(* IEC 61131-3 sources: AXOpen/src/showcase/app/src/ComponentsDukaneWelders/Documentation, 1 file *)

(* ---- DocumentationContext.st ---- *)
NAMESPACE AXOpen.Components.Dukane.Welders
    {S7.extern=ReadWrite}
    CLASS DocumentationContext EXTENDS AXOpen.Core.AxoObject
        VAR PUBLIC
            rootObject      : AxoObject;
            componentOne    : AXOpen.Components.Dukane.Welders.Component_1;
            componentTwo    : AXOpen.Components.Dukane.Welders.Component_2;
        END_VAR

        METHOD PUBLIC Execute
            rootObject.Run(THIS);
            componentOne.Run(rootObject);
            componentTwo.Run(rootObject);
        END_METHOD
    END_CLASS
END_NAMESPACE
